// TIA Portal V20 export
DATA_BLOCK "ShiftTimesList"   // DB52
TITLE = Shifttimes / Shift times
{ DB_Accessible_From_OPC_UA := 'FALSE' }
AUTHOR : SICAR
FAMILY : Shiftmodel
// Schichtzeiten Liste / Shift times List
// stored: DBAccessibleFromOPCUA false, MemoryReserve 100
   VAR
      list { ExternalAccessible := 'False'; ExternalVisible := 'False'; ExternalWritable := 'False'} : Array[0..10] of "LSicar_typeShiftmodTime1DaySel";   // Schichtmodel Liste / Shiftmodel list
   END_VAR
BEGIN
   list[3].listValidFor.sunday := TRUE;
   list[4].listValidFor.sunday := FALSE;
   list[1..3].listValidFor.monday := TRUE;
   list[4].listValidFor.monday := FALSE;
   list[1..3].listValidFor.tuesday := TRUE;
   list[4].listValidFor.tuesday := FALSE;
   list[1..3].listValidFor.wednesday := TRUE;
   list[4].listValidFor.wednesday := FALSE;
   list[1..3].listValidFor.thursday := TRUE;
   list[4].listValidFor.thursday := FALSE;
   list[1].listValidFor.friday := TRUE;
   list[3].listValidFor.friday := TRUE;
   list[4].listValidFor.friday := FALSE;
   list[3].listValidFor.saturday := TRUE;
   list[4].listValidFor.saturday := FALSE;
   list[1].shift[1].endCircuitTime := TOD#05:57:00;
   list[1].shift[2].endCircuitTime := TOD#13:57:00;
   list[1].shift[3].endCircuitTime := TOD#21:57:00;
   list[2].shift[1].endCircuitTime := TOD#04:57:00;
   list[2].shift[2].endCircuitTime := TOD#14:27:00;
   list[3].shift[1].endCircuitTime := TOD#05:57:00;
   list[3].shift[2].endCircuitTime := TOD#14:27:00;
   list[3].shift[3].endCircuitTime := TOD#22:57:00;
   list[4].shift[1..3].endCircuitTime := TOD#00:00:00;
   list[1].shift[1].start := TOD#06:00:00;
   list[1].shift[2].start := TOD#14:00:00;
   list[1].shift[3].start := TOD#22:00:00;
   list[2].shift[1].start := TOD#05:00:00;
   list[2].shift[2].start := TOD#14:30:00;
   list[3].shift[1].start := TOD#06:00:00;
   list[3].shift[2].start := TOD#14:30:00;
   list[3].shift[3].start := TOD#23:00:00;
   list[4].shift[1..3].start := TOD#00:00:00;
   list[1].shift[1].break[1].start := TOD#08:00:00;
   list[1].shift[1].break[2].start := TOD#10:00:00;
   list[1].shift[1].break[3].start := TOD#12:00:00;
   list[1].shift[1].break[4].start := TOD#00:00:00;
   list[1].shift[2].break[1].start := TOD#16:00:00;
   list[1].shift[2].break[2].start := TOD#18:00:00;
   list[1].shift[2].break[3].start := TOD#20:00:00;
   list[1].shift[3].break[1].start := TOD#00:00:00;
   list[1].shift[3].break[2].start := TOD#02:00:00;
   list[1].shift[3].break[3].start := TOD#04:00:00;
   list[2].shift[1].break[1].start := TOD#07:00:00;
   list[2].shift[1].break[2].start := TOD#09:00:00;
   list[2].shift[1].break[3].start := TOD#11:00:00;
   list[2].shift[1].break[4].start := TOD#13:00:00;
   list[2].shift[2].break[1].start := TOD#16:30:00;
   list[2].shift[2].break[2].start := TOD#18:30:00;
   list[2].shift[2].break[3].start := TOD#20:30:00;
   list[2].shift[2].break[4].start := TOD#22:00:00;
   list[3].shift[1].break[1].start := TOD#08:00:00;
   list[3].shift[1].break[2].start := TOD#10:00:00;
   list[3].shift[1].break[3].start := TOD#11:30:00;
   list[3].shift[1].break[4].start := TOD#12:30:00;
   list[3].shift[2].break[1].start := TOD#16:00:00;
   list[3].shift[2].break[2].start := TOD#18:00:00;
   list[3].shift[2].break[3].start := TOD#19:30:00;
   list[3].shift[2].break[4].start := TOD#20:30:00;
   list[3].shift[3].break[1].start := TOD#00:00:00;
   list[3].shift[3].break[2].start := TOD#02:00:00;
   list[3].shift[3].break[3].start := TOD#03:30:00;
   list[3].shift[3].break[4].start := TOD#04:30:00;
   list[4].shift[1].break[1..4].start := TOD#00:00:00;
   list[4].shift[2].break[1..4].start := TOD#00:00:00;
   list[4].shift[3].break[1..4].start := TOD#00:00:00;
   list[1].shift[1].break[1].startCircuitTime := TOD#08:02:00;
   list[1].shift[1].break[2].startCircuitTime := TOD#00:00:00;
   list[1].shift[1].break[3].startCircuitTime := TOD#12:02:00;
   list[1].shift[1].break[4].startCircuitTime := TOD#00:00:00;
   list[1].shift[2].break[1].startCircuitTime := TOD#16:02:00;
   list[1].shift[2].break[2].startCircuitTime := TOD#00:00:00;
   list[1].shift[2].break[3].startCircuitTime := TOD#20:02:00;
   list[1].shift[3].break[1].startCircuitTime := TOD#00:02:00;
   list[1].shift[3].break[2].startCircuitTime := TOD#00:00:00;
   list[1].shift[3].break[3].startCircuitTime := TOD#04:02:00;
   list[2].shift[1].break[1].startCircuitTime := TOD#07:02:00;
   list[2].shift[1].break[2].startCircuitTime := TOD#00:00:00;
   list[2].shift[1].break[3].startCircuitTime := TOD#11:02:00;
   list[2].shift[1].break[4].startCircuitTime := TOD#13:02:00;
   list[2].shift[2].break[1].startCircuitTime := TOD#16:32:00;
   list[2].shift[2].break[2].startCircuitTime := TOD#00:00:00;
   list[2].shift[2].break[3].startCircuitTime := TOD#20:32:00;
   list[2].shift[2].break[4].startCircuitTime := TOD#22:02:00;
   list[3].shift[1].break[1].startCircuitTime := TOD#00:00:00;
   list[3].shift[1].break[2].startCircuitTime := TOD#10:02:00;
   list[3].shift[1].break[3].startCircuitTime := TOD#00:00:00;
   list[3].shift[1].break[4].startCircuitTime := TOD#12:32:00;
   list[3].shift[2].break[1].startCircuitTime := TOD#00:00:00;
   list[3].shift[2].break[2].startCircuitTime := TOD#18:02:00;
   list[3].shift[2].break[3].startCircuitTime := TOD#00:00:00;
   list[3].shift[2].break[4].startCircuitTime := TOD#20:32:00;
   list[3].shift[3].break[1].startCircuitTime := TOD#00:00:00;
   list[3].shift[3].break[2].startCircuitTime := TOD#02:02:00;
   list[3].shift[3].break[3..4].startCircuitTime := TOD#00:00:00;
   list[4].shift[1].break[1..4].startCircuitTime := TOD#00:00:00;
   list[4].shift[2].break[1..4].startCircuitTime := TOD#00:00:00;
   list[4].shift[3].break[1..4].startCircuitTime := TOD#00:00:00;
   list[1].shift[1].break[1].endCircuitTime := TOD#08:13:00;
   list[1].shift[1].break[2].endCircuitTime := TOD#00:00:00;
   list[1].shift[1].break[3].endCircuitTime := TOD#12:13:00;
   list[1].shift[1].break[4].endCircuitTime := TOD#00:00:00;
   list[1].shift[2].break[1].endCircuitTime := TOD#16:13:00;
   list[1].shift[2].break[2].endCircuitTime := TOD#00:00:00;
   list[1].shift[2].break[3].endCircuitTime := TOD#20:13:00;
   list[1].shift[3].break[1].endCircuitTime := TOD#00:13:00;
   list[1].shift[3].break[2].endCircuitTime := TOD#00:00:00;
   list[1].shift[3].break[3].endCircuitTime := TOD#04:13:00;
   list[2].shift[1].break[1].endCircuitTime := TOD#07:13:00;
   list[2].shift[1].break[2].endCircuitTime := TOD#00:00:00;
   list[2].shift[1].break[3].endCircuitTime := TOD#11:13:00;
   list[2].shift[1].break[4].endCircuitTime := TOD#13:13:00;
   list[2].shift[2].break[1].endCircuitTime := TOD#16:43:00;
   list[2].shift[2].break[2].endCircuitTime := TOD#00:00:00;
   list[2].shift[2].break[3].endCircuitTime := TOD#20:43:00;
   list[2].shift[2].break[4].endCircuitTime := TOD#22:13:00;
   list[3].shift[1].break[1].endCircuitTime := TOD#00:00:00;
   list[3].shift[1].break[2].endCircuitTime := TOD#10:13:00;
   list[3].shift[1].break[3].endCircuitTime := TOD#00:00:00;
   list[3].shift[1].break[4].endCircuitTime := TOD#12:43:00;
   list[3].shift[2].break[1].endCircuitTime := TOD#00:00:00;
   list[3].shift[2].break[2].endCircuitTime := TOD#18:13:00;
   list[3].shift[2].break[3].endCircuitTime := TOD#00:00:00;
   list[3].shift[2].break[4].endCircuitTime := TOD#20:43:00;
   list[3].shift[3].break[1].endCircuitTime := TOD#00:00:00;
   list[3].shift[3].break[2].endCircuitTime := TOD#02:13:00;
   list[3].shift[3].break[3..4].endCircuitTime := TOD#00:00:00;
   list[4].shift[1].break[1..4].endCircuitTime := TOD#00:00:00;
   list[4].shift[2].break[1..4].endCircuitTime := TOD#00:00:00;
   list[4].shift[3].break[1..4].endCircuitTime := TOD#00:00:00;
   list[1].shift[1].break[1].end := TOD#08:15:00;
   list[1].shift[1].break[2].end := TOD#10:10:00;
   list[1].shift[1].break[3].end := TOD#12:15:00;
   list[1].shift[1].break[4].end := TOD#00:00:00;
   list[1].shift[2].break[1].end := TOD#16:15:00;
   list[1].shift[2].break[2].end := TOD#18:10:00;
   list[1].shift[2].break[3].end := TOD#20:15:00;
   list[1].shift[3].break[1].end := TOD#00:15:00;
   list[1].shift[3].break[2].end := TOD#02:10:00;
   list[1].shift[3].break[3].end := TOD#04:15:00;
   list[2].shift[1].break[1].end := TOD#07:15:00;
   list[2].shift[1].break[2].end := TOD#09:10:00;
   list[2].shift[1].break[3].end := TOD#11:15:00;
   list[2].shift[1].break[4].end := TOD#13:15:00;
   list[2].shift[2].break[1].end := TOD#16:45:00;
   list[2].shift[2].break[2].end := TOD#18:40:00;
   list[2].shift[2].break[3].end := TOD#20:45:00;
   list[2].shift[2].break[4].end := TOD#22:15:00;
   list[3].shift[1].break[1].end := TOD#08:10:00;
   list[3].shift[1].break[2].end := TOD#10:15:00;
   list[3].shift[1].break[3].end := TOD#11:40:00;
   list[3].shift[1].break[4].end := TOD#12:45:00;
   list[3].shift[2].break[1].end := TOD#16:10:00;
   list[3].shift[2].break[2].end := TOD#18:15:00;
   list[3].shift[2].break[3].end := TOD#19:40:00;
   list[3].shift[2].break[4].end := TOD#20:45:00;
   list[3].shift[3].break[1].end := TOD#00:10:00;
   list[3].shift[3].break[2].end := TOD#02:15:00;
   list[3].shift[3].break[3].end := TOD#03:40:00;
   list[3].shift[3].break[4].end := TOD#04:45:00;
   list[4].shift[1].break[1..4].end := TOD#00:00:00;
   list[4].shift[2].break[1..4].end := TOD#00:00:00;
   list[4].shift[3].break[1..4].end := TOD#00:00:00;
   list[1].shift[1].end := TOD#13:30:00;
   list[1].shift[2].end := TOD#21:30:00;
   list[1].shift[3].end := TOD#05:30:00;
   list[2].shift[1].end := TOD#14:00:00;
   list[2].shift[2].end := TOD#23:30:00;
   list[3].shift[1].end := TOD#13:30:00;
   list[3].shift[2].end := TOD#21:30:00;
   list[3].shift[3].end := TOD#05:30:00;
   list[4].shift[1..3].end := TOD#00:00:00;
   list[1].shift[1].startCircuitTime := TOD#13:33:00;
   list[1].shift[2].startCircuitTime := TOD#21:33:00;
   list[1].shift[3].startCircuitTime := TOD#05:33:00;
   list[2].shift[1].startCircuitTime := TOD#14:03:00;
   list[2].shift[2].startCircuitTime := TOD#23:33:00;
   list[3].shift[1].startCircuitTime := TOD#13:33:00;
   list[3].shift[2].startCircuitTime := TOD#21:33:00;
   list[3].shift[3].startCircuitTime := TOD#05:33:00;
   list[4].shift[1..3].startCircuitTime := TOD#00:00:00;
END_DATA_BLOCK
